KUKA KRL data list: PROCESSLOOP.dat

&ACCESS RVP
&REL 4
DEFDAT PROCESSLOOP PUBLIC

DECL CHAR MSG
DECL CHAR STATE
DECL E6POS MyPos
DECL BOOL MyBool
DECL BOOL AVAILABLE

ENDDAT
